# EPICS substitutions: IOCs/12id/iocBoot/ioc12ida1/softMotor.substitutions
file "$(STD)/stdApp/Db/softMotor.db"
{
pattern
{P,		SM}
{12ida1:,	SM1}
{12ida1:,	SM2}
{12ida1:,	SM3}
{12ida1:,	SM4}
{12ida1:,	SM5}
{12ida1:,	SM6}
{12ida1:,	SM7}
{12ida1:,	SM8}
{12ida1:,	SM9}
{12ida1:,	SM10}
{12ida1:,	dummy}
}
